// TIA Portal V20 export
DATA_BLOCK "SP203"   // DB346
// stored: MemoryReserve 100
   VAR
      "MODE SELECT AUTO" : Bool := FALSE;
      "HOME PBL (GREEN)" : Bool := FALSE;
      "SAFETY RESET PBL (BLUE)" : Bool := FALSE;
      "SCS MODE SELECT AUTO" : Bool := FALSE;
      "MODE SELECT MANUAL" : Bool := TRUE;
      "ENABLE PBL (BLACK)" : Bool := FALSE;
      "SCS MODE SELECT SETUP" : Bool := TRUE;
      "SCS MODE SELECT DISABLE" : Bool := FALSE;
   END_VAR
BEGIN
END_DATA_BLOCK
